# EPICS substitutions: SoftRamplcApp/Db/coils.substitutions
file "ramp.template"
{
    pattern { ORIENTATION, HW_SP }
            { H,           "PS-LCH-1:" }
            { V,           "PS-LCV:" }
}
